FUNCTION_BLOCK FB_EthDevice
VAR_INPUT
	bEnable		: BOOL 			:= FALSE;				(* TRUE => enable client data exchange, FALSE => disable *)
	sSrvNetID	: T_AmsNetID	:= '';					(* TwinCAT TCP/IP server network address *)
	sRemoteHost	: T_IPv4Addr 	:= '127.0.0.1';			(* Server network address *)
	nRemotePort	: UDINT 		:= 200;					(* Server port number *)
	bLogEnable	: BOOL 			:= FALSE;				(* TRUE => Enable log message output, FALSE => Disable *)
	sLogPrefix	: STRING 		:= 'CLIENT::';			(* Log message description string (allows the identification of log message source) *)
END_VAR
VAR_OUTPUT
	sData						: T_MaxString;			(* Output received Data *)
	bConnected					: BOOL := FALSE;		(* TCP/IP connection state *)	
END_VAR
VAR
	fbConnection				: FB_ClientConnection;	(* Client connection/data exchange control function block *)
	fbTx 						: FB_FrameFifo;			(* Tx fifo *)
	fbRx 						: FB_FrameFifo;			(* Rx fifo *)
	
	sLogMessage					: T_MaxString;
	sTemData					: T_MaxString;			(* Output received Data *)
END_VAR

IF bConnected := fbConnection.bConnected THEN
	A_Receive();
END_IF

A_Call();

IF NOT fbConnection.RxBusy THEN
	sData := sTemData;
END_IF

ACTION A_Call:
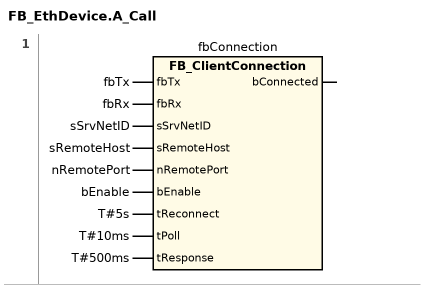
// NETWORK 1
fbConnection(
    fbTx := fbTx,
    fbRx := fbRx,
    sSrvNetID := sSrvNetID,
    sRemoteHost := sRemoteHost,
    nRemotePort := nRemotePort,
    bEnable := bEnable,
    tReconnect := T#5s,
    tPoll := T#10ms,
    tResponse := T#500ms); // FB_ClientConnection
END_ACTION

ACTION A_Receive:
	(*--------------------- Get received message strings --------------------------------*)
	REPEAT
		fbRx.RemoveHead( );(* Fetch string from rx fifo *)
		IF fbRx.bOk THEN(* Success *)
	
		(* TODO: Implement receive data handler *)
			sTemData := fbRx.sGet; 		
			
		END_IF
	UNTIL NOT fbRx.bOk
	END_REPEAT
END_ACTION

METHOD Send : BOOL
VAR_INPUT
	sTxData		: T_MaxString;	(* Data to send *)
END_VAR
VAR
	RTRIG_SendCommand			: R_TRIG;
END_VAR
		fbTx.AddTail( sPut := sTxData );(* Put string to the tx fifo *)
END_METHOD

END_FUNCTION_BLOCK

(* stored: Version 1.1.0.1, ProductVersion 3.1.4024.13
   POU FB_EthDevice: Id {c11f7280-27ca-4f3d-865b-a554dd255326}, SpecialFunc None
   Action A_Call: Id {9bbcadd1-063f-4649-8065-66483265221a}
   Action A_Receive: Id {44b562d5-7166-4ed6-8902-d98806e6705c}
   Method Send: Id {6d0fdf11-2b9c-45c0-94d0-44e8e8ce1a4f} *)
